// TIA Portal V17 export
// export: Created 2023-12-22T15:05:28.546595Z, ExportSetting WithDefaults, DisplayName Totally Integrated Automation Portal, DisplayVersion V17, DisplayName TIA Portal Openness, DisplayVersion V17, DisplayName TIA Portal Version Control Interface, DisplayVersion V17, DisplayName STEP 7 Professional, DisplayVersion V17, DisplayName STEP 7 Safety, DisplayVersion V17, DisplayName WinCC Advanced, DisplayVersion V17
FUNCTION_BLOCK "AOx"   // FB230, LAD
TITLE = Регулируемые устройства
{ S7_Optimized_Access := 'FALSE' }
VERSION : 0.1
// SP - управляющий сигнал из программы, формат Real
// Signal - PQW код выходного сигнала контроллера
// stored: AutoNumber false, IsIECCheckEnabled false, SetENOAutomatically false, UDAEnableTagReadback false
   VAR DB_SPECIFIC
      Time_DTL { S7_SetPoint := 'True'} : DTL;
   END_VAR
BEGIN

REGION Network 1: Example
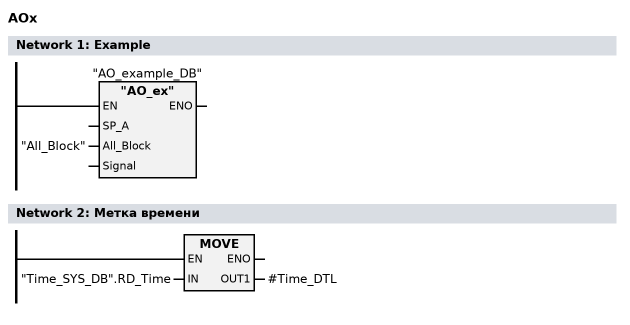
   RUNG wire#powerrail
      "AO_example_DB"(SP_A :=, All_Block := "All_Block", Signal :=)
   END_RUNG
   // the same network as SCL:
   "AO_example_DB"(All_Block := "All_Block");   // "AO_ex"
END_REGION

REGION Network 2: Метка времени
   RUNG wire#powerrail
      Move(in := "Time_SYS_DB".RD_Time, out1 => #Time_DTL)
   END_RUNG
   // the same network as SCL:
   #Time_DTL := "Time_SYS_DB".RD_Time;
END_REGION
END_FUNCTION_BLOCK
